// TIA Portal V20 export
TYPE "LConSMC_typeWebbreakDetectConfig"
// Konfiguration der Bahnrisserkennung / Configuration parameters for webbreak detection
// stored: Access Published
   STRUCT
      enableDetection : Bool;   // TRUE: Freigabe der Bahnrissüberwachung / TRUE: Enable webbreak detection
      minLineVelocity : LReal;   // [m/min or ft/min] Minimale Bahngeschwindigkeit ab der die Überwachung aktiviert wird / [m/min or ft/min] Minimum line speed for detection to be active
      upperLimitError : LReal;   // [Einheit des Zug-/Tänzeristwertes] Oberere Grenzwert bei dem ein Bahnriss erkannt wird !Im Regelungmodus "Indirekte Zugregelung" wird die Soll-/Istdrehmomentabweichung bezogen auf das Referenzdrehmoment in Prozent überwacht! / [Unit of tension/dancer feedback] Upper limit for detecting web break !In the control mode "Indirect tension control" the torque deviation in relation to the reference torque in precent is monitored!
      lowerLimitError : LReal;   // [Einheit des Zug-/Tänzeristwertes] Unterer Grenzwert bei dem ein Bahnriss erkannt wird !Im Regelungmodus "Indirekte Zugregelung" wird die Soll-/Istdrehmomentabweichung bezogen auf das Referenzdrehmoment in Prozent überwacht! / [Unit of tension/dancer feedback] Lower limit for detecting web break !In the control mode "Indirect tension control" the torque deviation in relation to the reference torque in precent is monitored!
      delayTime : Time;   // Verzögerungszeit nachdem der Diagoseausgang "webBreak" = TRUE gesetzt wird / Delay time before diagnostic output "webBreak" is set to TRUE
   END_STRUCT;
END_TYPE
